(* IEC 61131-3 sources: Std_PalletMover/Class/RiwoAlarmCollect, 1 file *)

(* ---- RiwoAlarmCollect.st ---- *)
(*!
<Class
	Name               = "RiwoAlarmCollect"
	Revision           = "0.1"
	RealtimeTask       = "false"
	CyclicTask         = "false"
	BackgroundTask     = "true"
	DefBackground      = "100 ms"
	Sigmatek           = "false"
	OSInterface        = "false"
	HighPriority       = "false"
	Automatic          = "false"
	UpdateMode         = "Prescan"
	SharedCommandTable = "true"
	Objectsize         = "(738,120)">
	<Channels>
		<Server Name="ClassSvr" Visualized="false" Initialize="false" WriteProtected="true" Retentive="false"/>
		<Server Name="ErrorReportConfig" Visualized="true" Initialize="false" WriteProtected="true" Retentive="false"/>
		<Server Name="Errors" Visualized="true" Initialize="false" WriteProtected="true" Retentive="false"/>
		<Server Name="Warnings" Visualized="true" Initialize="false" WriteProtected="true" Retentive="false"/>
		<Client Name="objFirstRiwoParamAlarm" Required="false" Internal="false"/>
	</Channels>
	<Dependencies>
		<Files>
			<File Path=".\Class\RiwoDefine\RiwoDef.h" Include="false"/>
		</Files>
	</Dependencies>
</Class>
*)
RiwoAlarmCollect : CLASS
  //Servers:
	ClassSvr 	: SvrChCmd_DINT;
	Errors 	: SvrCh_BDINT;
	Warnings 	: SvrCh_BDINT;
	ErrorReportConfig 	: SvrCh_BDINT;
  //Clients:
	objFirstRiwoParamAlarm 	: CltChCmd_RiwoParamAlarm;
  //Variables:
  //Functions:

	FUNCTION VIRTUAL GLOBAL Background
		VAR_INPUT
			EAX 	: UDINT;
		END_VAR
		VAR_OUTPUT
			state (EAX) 	: UDINT;
		END_VAR;
  //Tables:
	FUNCTION @STD
		VAR_OUTPUT
			ret_code	: CONFSTATES;
		END_VAR;
	FUNCTION GLOBAL TAB @CT_;
END_CLASS;

#pragma usingLtd RiwoParamAlarm

//handle getting the data from the connecte errors
FUNCTION VIRTUAL GLOBAL RiwoAlarmCollect::Background
	VAR_INPUT
		EAX 	: UDINT;
	END_VAR
	VAR_OUTPUT
		state (EAX) 	: UDINT;
	END_VAR

	state := READY;

  if IsClientConnected(input:= #objFirstRiwoParamAlarm) = true then
    Errors := objFirstRiwoParamAlarm.GetActiveErrors(objNr:= 0);
    Errors.Write(input:= Errors);
    Warnings := objFirstRiwoParamAlarm.GetActiveWarnings(objNr:= 0);
    Warnings.Write(input:=Warnings);
    ErrorReportConfig := objFirstRiwoParamAlarm.GetReportConfigs(objNr:=0);
    ErrorReportConfig.Write(input:=ErrorReportConfig);
  end_if;

END_FUNCTION
